{attribute addProperty BoxType "EK1122-0000-0018"}
{attribute addProperty Id "Beckhoff_EP3xxxsub_EK1100EK1100_179A0949162A_0001_EP3162_0002_0016EP3162_1C870F0C16020A_0002_EP3162_1002_0017EP3162_461C4AB617622A_0003_EP3174_0002_0016EP3174_8D19A6A542052.5A_0004_EP3174_0002_0017EP3174_8D19A6A542052.5A_0005_EP3174_0002_0018EP3174_55F04E9922428A_0006_EP3174_0002_0019EP3174_55F04E9922428A_0007_EP3174_0002_0020EP3174_83515A0D22428A_0008_EP3174_0002_0021EP3174_83515A0D22428A_0009_EP3174_0002_0022EP3174_83515A0D22428A_0010_EP3174_0002_0023EP3174_83515A0D22428A_0011_EP3174_0092_0016EP3174_83515A0D22428A_0012_EP3182_1002_0017EP3182_E7AA79FE17622A_0013_EP3182_1002_0018EP3182_461C4AB617622A_0014_EP3182_1002_0019EP3182_461C4AB617622A_0015_EP3182_1002_0020EP3182_461C4AB617622A_0016_EP3184_0002_0016EP3184_8D19A6A542052.5A_0017_EP3184_0002_0017EP3184_55F04E9922428A_0018_EP3184_0002_0018EP3184_55F04E9922428A_0019_EP3184_0002_0019EP3184_55F04E9922428A_0020_EP3184_0002_0020EP3184_55F04E9922428A_0021_EP3184_0002_0021EP3184_83515A0D22428A_0022_EP3184_0402_0016EP3184_55F04E9922428A_0023_EP3184_0402_0017EP3184_55F04E9922428A_0024_EP3184_0402_0018EP3184_83515A0D22428A_0025_EP3184_1002_0016EP3184_8D19A6A542052.5A_0026_EP3184_1002_0017EP3184_8D19A6A542052.5A_0027_EP3184_1002_0018EP3184_55F04E9922428A_0028_EP3184_1002_0019EP3184_55F04E9922428A_0029_EP3184_1002_0020EP3184_55F04E9922428A_0030_EP3184_1002_0021EP3184_83515A0D22428A_0031_EP3204_0002_0017EP3204_BF093E1239249A_0032_EP3204_0002_0018EP3204_BF093E1239249A_0033_EP3204_0002_0019EP3204_BF093E1239249A_0034_EP3204_0002_0020EP3204_BF093E1239249A_0035_EP3204_0002_0021EP3204_69AA4F8E22428A_0036_EP3314_0002_0016EP3314_7758490939249A_0037_EP3314_0002_0017EP3314_7758490939249A_0038_EP3314_0002_0018EP3314_AF8E369F22428A_0039_EP3314_0002_0019EP3314_2E54E3B022428A_0040_EP3314_0002_0020EP3314_2E54E3B022428A_0041_EP3314_0002_0021EP3314_2E54E3B022428A_0042_EP3351_2022_0016EP3351_606039E324030A_0043_EP3356_0022_0016EP3356_CA56400F16020A_0044_EP3356_0022_0017EP3356_CA56400F16020A_0045_EP3356_0022_0022EP3356_CA56400F16020A_0046_EP3632_0001_0016EP3632_C340233D59274A_0047_EP3632_0001_0017EP3632_C340233D59274A_0048_EP3744_0041_0016EP3744_38AF8BFB40050A_0049_EP3744_0041_0017EP3744_38AF8BFB40050A_0050_EP3744_0041_0018EP3744_38AF8BFB40050A_0051_EP3744_0041_0019EP3744_38AF8BFB40050A_0052_EP3744_0041_0020EP3744_38AF8BFB40050A_0053_EP3744_0041_0021EP3744_38AF8BFB40050A_0054_EP3744_1041_0016EP3744_38AF8BFB40050A_0055_EP3744_1041_0017EP3744_38AF8BFB40050A_0056_EP3744_1041_0018EP3744_38AF8BFB40050A_0057_EP3744_1041_0019EP3744_38AF8BFB40050A_0058_EP3744_1041_0020EP3744_38AF8BFB40050A_0059_EP3744_1041_0021EP3744_38AF8BFB40050A_0060_EP3752_0000_0017EP3752_AEF24F9C28836A_0061_EP3752_0000_0018EP3752_AEF24F9C28836"}
{attribute addProperty CRC "1311078606"}
{attribute addProperty SizeInBites "18164"}
{attribute addProperty SizeInBytes "2270.5"}
TYPE Beckhoff_EP3xxxEK1122_4E2578CE EXTENDS EK1122_179A0949 :
STRUCT
	{attribute addProperty Name "Beckhoff_EP3xxxsub_EK1100"}
	Beckhoff_EP3xxxsub_EK1100 : EK1100_179A0949;
	{attribute addProperty Name "A_0001_EP3162_0002_0016"}
	A_0001_EP3162_0002_0016 : EP3162_1C870F0C;
	{attribute addProperty Name "A_0002_EP3162_1002_0017"}
	A_0002_EP3162_1002_0017 : EP3162_461C4AB6;
	{attribute addProperty Name "A_0003_EP3174_0002_0016"}
	A_0003_EP3174_0002_0016 : EP3174_8D19A6A5;
	{attribute addProperty Name "A_0004_EP3174_0002_0017"}
	A_0004_EP3174_0002_0017 : EP3174_8D19A6A5;
	{attribute addProperty Name "A_0005_EP3174_0002_0018"}
	A_0005_EP3174_0002_0018 : EP3174_55F04E99;
	{attribute addProperty Name "A_0006_EP3174_0002_0019"}
	A_0006_EP3174_0002_0019 : EP3174_55F04E99;
	{attribute addProperty Name "A_0007_EP3174_0002_0020"}
	A_0007_EP3174_0002_0020 : EP3174_83515A0D;
	{attribute addProperty Name "A_0008_EP3174_0002_0021"}
	A_0008_EP3174_0002_0021 : EP3174_83515A0D;
	{attribute addProperty Name "A_0009_EP3174_0002_0022"}
	A_0009_EP3174_0002_0022 : EP3174_83515A0D;
	{attribute addProperty Name "A_0010_EP3174_0002_0023"}
	A_0010_EP3174_0002_0023 : EP3174_83515A0D;
	{attribute addProperty Name "A_0011_EP3174_0092_0016"}
	A_0011_EP3174_0092_0016 : EP3174_83515A0D;
	{attribute addProperty Name "A_0012_EP3182_1002_0017"}
	A_0012_EP3182_1002_0017 : EP3182_E7AA79FE;
	{attribute addProperty Name "A_0013_EP3182_1002_0018"}
	A_0013_EP3182_1002_0018 : EP3182_461C4AB6;
	{attribute addProperty Name "A_0014_EP3182_1002_0019"}
	A_0014_EP3182_1002_0019 : EP3182_461C4AB6;
	{attribute addProperty Name "A_0015_EP3182_1002_0020"}
	A_0015_EP3182_1002_0020 : EP3182_461C4AB6;
	{attribute addProperty Name "A_0016_EP3184_0002_0016"}
	A_0016_EP3184_0002_0016 : EP3184_8D19A6A5;
	{attribute addProperty Name "A_0017_EP3184_0002_0017"}
	A_0017_EP3184_0002_0017 : EP3184_55F04E99;
	{attribute addProperty Name "A_0018_EP3184_0002_0018"}
	A_0018_EP3184_0002_0018 : EP3184_55F04E99;
	{attribute addProperty Name "A_0019_EP3184_0002_0019"}
	A_0019_EP3184_0002_0019 : EP3184_55F04E99;
	{attribute addProperty Name "A_0020_EP3184_0002_0020"}
	A_0020_EP3184_0002_0020 : EP3184_55F04E99;
	{attribute addProperty Name "A_0021_EP3184_0002_0021"}
	A_0021_EP3184_0002_0021 : EP3184_83515A0D;
	{attribute addProperty Name "A_0022_EP3184_0402_0016"}
	A_0022_EP3184_0402_0016 : EP3184_55F04E99;
	{attribute addProperty Name "A_0023_EP3184_0402_0017"}
	A_0023_EP3184_0402_0017 : EP3184_55F04E99;
	{attribute addProperty Name "A_0024_EP3184_0402_0018"}
	A_0024_EP3184_0402_0018 : EP3184_83515A0D;
	{attribute addProperty Name "A_0025_EP3184_1002_0016"}
	A_0025_EP3184_1002_0016 : EP3184_8D19A6A5;
	{attribute addProperty Name "A_0026_EP3184_1002_0017"}
	A_0026_EP3184_1002_0017 : EP3184_8D19A6A5;
	{attribute addProperty Name "A_0027_EP3184_1002_0018"}
	A_0027_EP3184_1002_0018 : EP3184_55F04E99;
	{attribute addProperty Name "A_0028_EP3184_1002_0019"}
	A_0028_EP3184_1002_0019 : EP3184_55F04E99;
	{attribute addProperty Name "A_0029_EP3184_1002_0020"}
	A_0029_EP3184_1002_0020 : EP3184_55F04E99;
	{attribute addProperty Name "A_0030_EP3184_1002_0021"}
	A_0030_EP3184_1002_0021 : EP3184_83515A0D;
	{attribute addProperty Name "A_0031_EP3204_0002_0017"}
	A_0031_EP3204_0002_0017 : EP3204_BF093E12;
	{attribute addProperty Name "A_0032_EP3204_0002_0018"}
	A_0032_EP3204_0002_0018 : EP3204_BF093E12;
	{attribute addProperty Name "A_0033_EP3204_0002_0019"}
	A_0033_EP3204_0002_0019 : EP3204_BF093E12;
	{attribute addProperty Name "A_0034_EP3204_0002_0020"}
	A_0034_EP3204_0002_0020 : EP3204_BF093E12;
	{attribute addProperty Name "A_0035_EP3204_0002_0021"}
	A_0035_EP3204_0002_0021 : EP3204_69AA4F8E;
	{attribute addProperty Name "A_0036_EP3314_0002_0016"}
	A_0036_EP3314_0002_0016 : EP3314_77584909;
	{attribute addProperty Name "A_0037_EP3314_0002_0017"}
	A_0037_EP3314_0002_0017 : EP3314_77584909;
	{attribute addProperty Name "A_0038_EP3314_0002_0018"}
	A_0038_EP3314_0002_0018 : EP3314_AF8E369F;
	{attribute addProperty Name "A_0039_EP3314_0002_0019"}
	A_0039_EP3314_0002_0019 : EP3314_2E54E3B0;
	{attribute addProperty Name "A_0040_EP3314_0002_0020"}
	A_0040_EP3314_0002_0020 : EP3314_2E54E3B0;
	{attribute addProperty Name "A_0041_EP3314_0002_0021"}
	A_0041_EP3314_0002_0021 : EP3314_2E54E3B0;
	{attribute addProperty Name "A_0042_EP3351_2022_0016"}
	A_0042_EP3351_2022_0016 : EP3351_606039E3;
	{attribute addProperty Name "A_0043_EP3356_0022_0016"}
	A_0043_EP3356_0022_0016 : EP3356_CA56400F;
	{attribute addProperty Name "A_0044_EP3356_0022_0017"}
	A_0044_EP3356_0022_0017 : EP3356_CA56400F;
	{attribute addProperty Name "A_0045_EP3356_0022_0022"}
	A_0045_EP3356_0022_0022 : EP3356_CA56400F;
	{attribute addProperty Name "A_0046_EP3632_0001_0016"}
	A_0046_EP3632_0001_0016 : EP3632_C340233D;
	{attribute addProperty Name "A_0047_EP3632_0001_0017"}
	A_0047_EP3632_0001_0017 : EP3632_C340233D;
	{attribute addProperty Name "A_0048_EP3744_0041_0016"}
	A_0048_EP3744_0041_0016 : EP3744_38AF8BFB;
	{attribute addProperty Name "A_0049_EP3744_0041_0017"}
	A_0049_EP3744_0041_0017 : EP3744_38AF8BFB;
	{attribute addProperty Name "A_0050_EP3744_0041_0018"}
	A_0050_EP3744_0041_0018 : EP3744_38AF8BFB;
	{attribute addProperty Name "A_0051_EP3744_0041_0019"}
	A_0051_EP3744_0041_0019 : EP3744_38AF8BFB;
	{attribute addProperty Name "A_0052_EP3744_0041_0020"}
	A_0052_EP3744_0041_0020 : EP3744_38AF8BFB;
	{attribute addProperty Name "A_0053_EP3744_0041_0021"}
	A_0053_EP3744_0041_0021 : EP3744_38AF8BFB;
	{attribute addProperty Name "A_0054_EP3744_1041_0016"}
	A_0054_EP3744_1041_0016 : EP3744_38AF8BFB;
	{attribute addProperty Name "A_0055_EP3744_1041_0017"}
	A_0055_EP3744_1041_0017 : EP3744_38AF8BFB;
	{attribute addProperty Name "A_0056_EP3744_1041_0018"}
	A_0056_EP3744_1041_0018 : EP3744_38AF8BFB;
	{attribute addProperty Name "A_0057_EP3744_1041_0019"}
	A_0057_EP3744_1041_0019 : EP3744_38AF8BFB;
	{attribute addProperty Name "A_0058_EP3744_1041_0020"}
	A_0058_EP3744_1041_0020 : EP3744_38AF8BFB;
	{attribute addProperty Name "A_0059_EP3744_1041_0021"}
	A_0059_EP3744_1041_0021 : EP3744_38AF8BFB;
	{attribute addProperty Name "A_0060_EP3752_0000_0017"}
	A_0060_EP3752_0000_0017 : EP3752_AEF24F9C;
	{attribute addProperty Name "A_0061_EP3752_0000_0018"}
	A_0061_EP3752_0000_0018 : EP3752_AEF24F9C;
END_STRUCT
END_TYPE

(* stored: Version 1.2.0.0, ProductVersion 3.1.4024.9
   DUT Beckhoff_EP3xxxEK1122_4E2578CE: Id {3520606d-4333-4567-b190-73fd69da5bc5} *)
